// TwinCAT 3 PLC project UDP
// ProgramVersion: 3.1.4020.2
// libraries:
//   Tc2_Standard, * (Beckhoff Automation GmbH)
//   Tc2_System, * (Beckhoff Automation GmbH)
//   Tc2_TcpIp, * (Beckhoff Automation GmbH)
//   Tc3_Module, * (Beckhoff Automation GmbH)
// project tree:
//   / PlcTask.TcTTO
//   POUs/ MAIN.TcPOU

CONFIGURATION UDP
    RESOURCE PLC ON TwinCAT3
        TASK PlcTask(INTERVAL := T#10ms, PRIORITY := 20);
        PROGRAM MAIN WITH PlcTask : MAIN;
    END_RESOURCE
END_CONFIGURATION

// ---- POUs/MAIN.TcPOU
PROGRAM MAIN
VAR
	fbSocketCreate	: FB_SocketUdpCreate;
	fbReceive		: FB_SocketUdpReceiveFrom;
	fbSend			: FB_SocketUdpSendTo;
	
	NetId: STRING := '';
	HostAdr: STRING := '127.0.0.1';
	Port: UDINT := 5005;
	hSocket: T_HSOCKET;
	
	sReceive : STRING;
	sSend : STRING := 'Neomuhae';
	
	
	
	
	fb1:FB_SocketConnect;
	fb2:FB_SocketReceive;
	fb3:FB_SocketSend;
END_VAR

fbSocketCreate(
	sSrvNetId:= NetId, 
	sLocalHost:= HostAdr, 
	nLocalPort:= Port, 
	bExecute:= , 
	tTimeout:= , 
	bBusy=> , 
	bError=> , 
	nErrId=> , 
	hSocket=> hSocket);
	
fbReceive(
	sSrvNetId:= NetId, 
	hSocket:= hSocket, 
	cbLen:= SIZEOF(sReceive), 
	pDest:= ADR(sReceive), 
	bExecute:= , 
	tTimeout:= , 
	bBusy=> , 
	bError=> , 
	nErrId=> , 
	sRemoteHost=> , 
	nRemotePort=> , 
	nRecBytes=> );
	
fbSend(
	sSrvNetId:= NetId, 
	hSocket:= hSocket, 
	sRemoteHost:= HostAdr, 
	nRemotePort:= Port, 
	cbLen:= LEN(sSend), 
	pSrc:= ADR(sSend), 
	bExecute:= , 
	tTimeout:= , 
	bBusy=> , 
	bError=> , 
	nErrId=> );
	
	
fb1(
	sSrvNetId:= NetId, 
	sRemoteHost:= HostAdr, 
	nRemotePort:= Port, 
	bExecute:= , 
	tTimeout:= , 
	bBusy=> , 
	bError=> , 
	nErrId=> , 
	hSocket=> hSocket);
	
fb2(
	sSrvNetId:= NetId, 
	hSocket:= hSocket, 
	cbLen:= SIZEOF(sReceive), 
	pDest:= ADR(sReceive), 
	bExecute:= , 
	tTimeout:= , 
	bBusy=> , 
	bError=> , 
	nErrId=> , 
	nRecBytes=> );
	
fb3(
	sSrvNetId:= NetId, 
	hSocket:= hSocket, 
	cbLen:= LEN(sSend), 
	pSrc:= ADR(sSend), 
	bExecute:= , 
	tTimeout:= , 
	bBusy=> , 
	bError=> , 
	nErrId=> );

END_PROGRAM
